(* LS Electric XG5000 project: TrafficLight *)
(* PLC LSPLC *)

FUNCTION_BLOCK GET_INT_REMAIN_TIME_SECOND
VAR_INPUT
    total_time : TIME;
    use_time : TIME;
END_VAR
VAR_OUTPUT
    result_time : INT;
END_VAR
VAR
    remian_time : TIME;
    str_result_time : STRING;
    str_time : STRING;
END_VAR

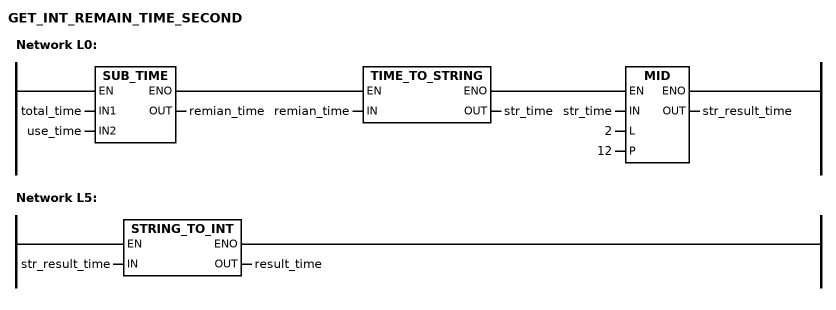
(* Rung L0 *)
remian_time := SUB_TIME(total_time, use_time);
str_time := TIME_TO_STRING(remian_time);
str_result_time := MID(IN := str_time, L := 2, P := 12);
(* Rung L5 *)
result_time := STRING_TO_INT(str_result_time);
END_FUNCTION_BLOCK

PROGRAM NewProgram (* task: 스캔 프로그램 *)
VAR
    flicker1 : FF;
    On_Button : BOOL;
    remain_time : GET_INT_REMAIN_TIME_SECOND;
    sequence0 : BOOL;
    sequence1 : BOOL;
    sequence2 : BOOL;
    sequence3 : BOOL;
    sequence4 : BOOL;
    sequence5 : BOOL;
    sequence6 : BOOL;
    str_remain_time : STRING;
    t10s : TON;
    t1s : TON;
    t30s : TON;
    t30s2 : TON;
    tof1 : TOF;
    tof2 : TOF;
    tof3 : TOF;
    tof4 : TOF;
    ton1 : TON;
    ton2 : TON;
    ton3 : TON;
    tp1 : TP;
    tp10s : TP;
    tp2 : TP;
    tp20s : TP;
    tp3 : TP;
    tp30s : TP;
    tp5s : TP;
    tp60 : TP;
    보행자_녹색불 AT %QX0.1.0 : BOOL;
    보행자_빨간불 AT %QX0.1.1 : BOOL;
    보행자_신호 AT %IX0.0.0 : BOOL;
    차량신호_노란불 AT %QX0.0.1 : BOOL;
    차량신호_녹색불 AT %QX0.0.2 : BOOL;
    차량신호_빨간불 AT %QX0.0.0 : BOOL;
END_VAR
VAR
    _p1 : BOOL;
    _p2 : BOOL;
END_VAR

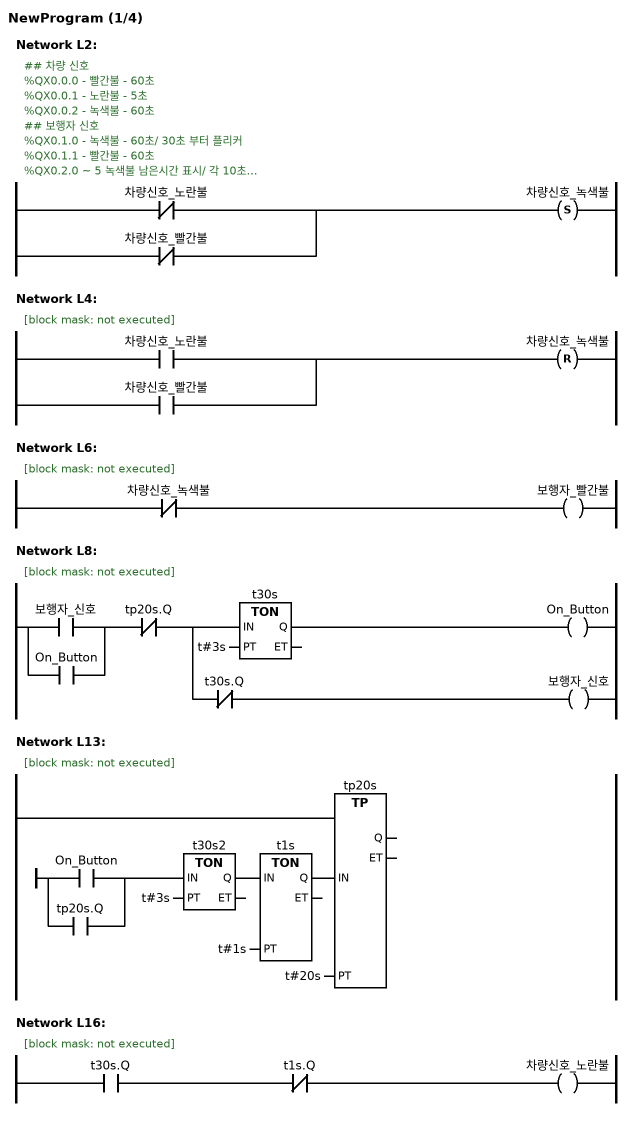
(* ## 차량 신호 / %QX0.0.0 - 빨간불 - 60초 / %QX0.0.1 - 노란불 - 5초 / %QX0.0.2 - 녹색불 - 60초 / ## 보행자 신호 / %QX0.1.0 - 녹색불 - 60초/ 30초 부터 플리커 / %QX0.1.1 - 빨간불 - 60초 / %QX0.2.0 ~ 5 녹색불 남은시간 표시/ 각 10초씩 *)
(* ## 차량신호 녹색불/ 보행자 신호 빨간불 유지 *)
(* Rung L2 is block-masked: not executed *)
// IF NOT 차량신호_노란불 OR NOT 차량신호_빨간불 THEN 차량신호_녹색불 := TRUE; END_IF;
(* Rung L4 is block-masked: not executed *)
// IF 차량신호_노란불 OR 차량신호_빨간불 THEN 차량신호_녹색불 := FALSE; END_IF;
(* Rung L6 is block-masked: not executed *)
// 보행자_빨간불 := NOT 차량신호_녹색불;
(* Rung L8 is block-masked: not executed *)
// t30s(IN := (보행자_신호 OR On_Button) AND NOT tp20s.Q, PT := t#3s);
// _p1 := (보행자_신호 OR On_Button) AND NOT tp20s.Q;
// On_Button := t30s.Q;
// 보행자_신호 := _p1 AND NOT t30s.Q;
(* Rung L13 is block-masked: not executed *)
// t30s2(IN := On_Button OR tp20s.Q, PT := t#3s);
// t1s(IN := t30s2.Q, PT := t#1s);
// tp20s(IN := t1s.Q, PT := t#20s);
(* Rung L16 is block-masked: not executed *)
// 차량신호_노란불 := t30s.Q AND NOT t1s.Q;

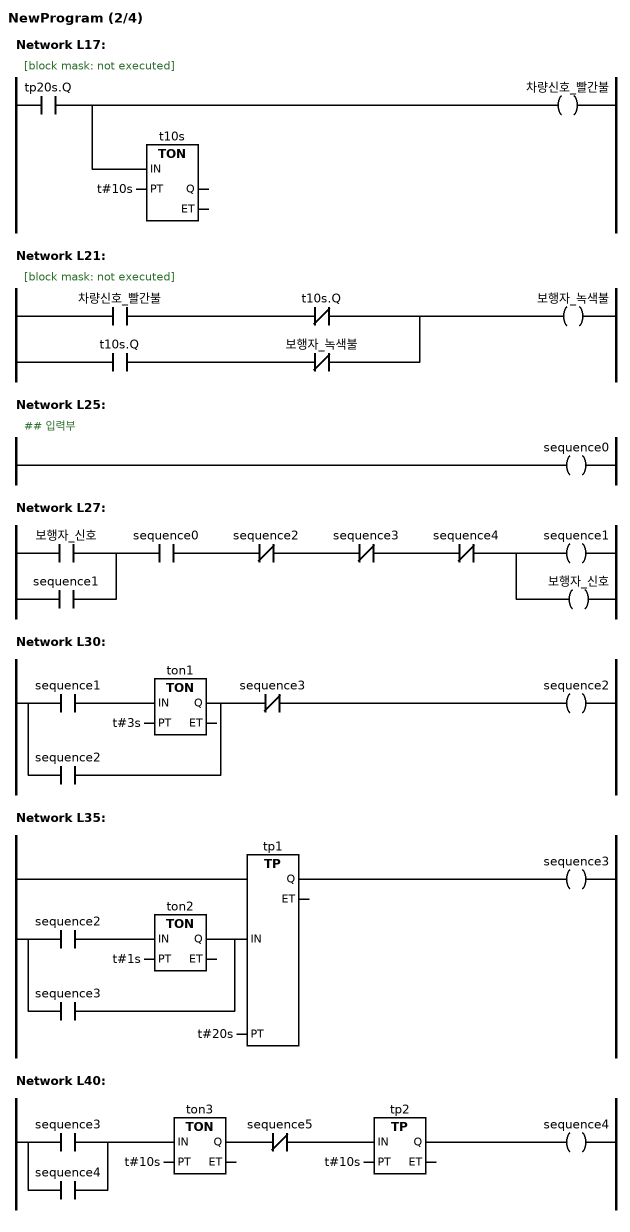
(* Rung L17 is block-masked: not executed *)
// 차량신호_빨간불 := tp20s.Q;
// t10s(IN := tp20s.Q, PT := t#10s);
(* Rung L21 is block-masked: not executed *)
// 보행자_녹색불 := (차량신호_빨간불 AND NOT t10s.Q) OR (t10s.Q AND NOT 보행자_녹색불);
(* ## 입력부 *)
(* Rung L25 *)
sequence0 := TRUE;
(* Rung L27 *)
_p2 := (보행자_신호 OR sequence1) AND sequence0 AND NOT sequence2 AND NOT sequence3 AND NOT sequence4;
sequence1 := _p2;
보행자_신호 := _p2;
(* Rung L30 *)
ton1(IN := sequence1, PT := t#3s);
sequence2 := (ton1.Q OR sequence2) AND NOT sequence3;
(* Rung L35 *)
ton2(IN := sequence2, PT := t#1s);
tp1(IN := ton2.Q OR sequence3, PT := t#20s);
sequence3 := tp1.Q;
(* Rung L40 *)
ton3(IN := sequence3 OR sequence4, PT := t#10s);
tp2(IN := ton3.Q AND NOT sequence5, PT := t#10s);
sequence4 := tp2.Q;

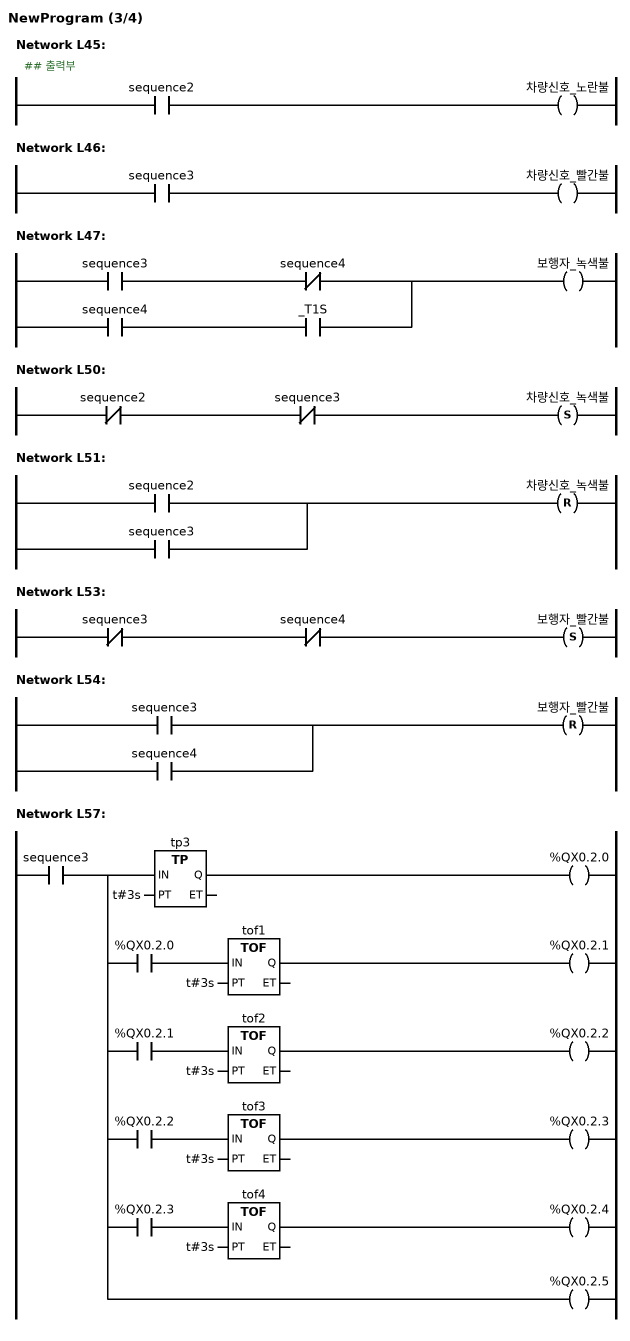
(* ## 출력부 *)
(* Rung L45 *)
차량신호_노란불 := sequence2;
(* Rung L46 *)
차량신호_빨간불 := sequence3;
(* Rung L47 *)
보행자_녹색불 := (sequence3 AND NOT sequence4) OR (sequence4 AND _T1S);
(* Rung L50 *)
IF NOT sequence2 AND NOT sequence3 THEN 차량신호_녹색불 := TRUE; END_IF;
(* Rung L51 *)
IF sequence2 OR sequence3 THEN 차량신호_녹색불 := FALSE; END_IF;
(* Rung L53 *)
IF NOT sequence3 AND NOT sequence4 THEN 보행자_빨간불 := TRUE; END_IF;
(* Rung L54 *)
IF sequence3 OR sequence4 THEN 보행자_빨간불 := FALSE; END_IF;
(* Rung L57 *)
tp3(IN := sequence3, PT := t#3s);
%QX0.2.0 := tp3.Q;
tof1(IN := sequence3 AND %QX0.2.0, PT := t#3s);
%QX0.2.1 := tof1.Q;
tof2(IN := sequence3 AND %QX0.2.1, PT := t#3s);
%QX0.2.2 := tof2.Q;
tof3(IN := sequence3 AND %QX0.2.2, PT := t#3s);
%QX0.2.3 := tof3.Q;
tof4(IN := sequence3 AND %QX0.2.3, PT := t#3s);
%QX0.2.4 := tof4.Q;
%QX0.2.5 := sequence3;

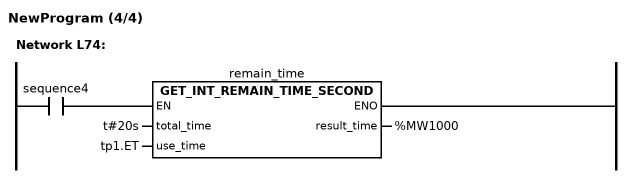
(* Rung L74 *)
IF sequence4 THEN remain_time(total_time := t#20s, use_time := tp1.ET, result_time => %MW1000); END_IF;
END_PROGRAM